TYPE ST_ITC_ZoneCommands :
(**************************************************************************************
 * 	Application		:	BoxControl Framework
 *	Revision		:	$Revision: 404529 $
 *	Revision date	:	$Date: 2018-04-23 08:21:38 +0200 (Mo., 23 Apr 2018) $
 *	Last changed by	:	$Author: b7bolm $
 *	URL				:	$URL: http://almscdc.swisslog.com/repo/SWPD/Development/BoxControlFramework/20_Release/trunk/01_Software/BCF/BCF/JumpStart/20_Product/10_App/12_E_Functions/10_Lib/10_Conv/01_DUTs/ST_ITC_ZoneCommands.TcDUT $
 *
 *	Purpose			:	Zone commands
 *
 * ------------------------------------------------------------------------------------
 *	Copyright Swisslog [IP AG], Switzerland. All rights reserved.
 * 
 * ------------------------------------------------------------------------------------
 *	
 * 	Revision History: 
 *
 * 	VERSION			DATE			INITIALS			DESCRIPTION
 *	0.1				01.01.2001		swl					Example
 *
 **************************************************************************************)	
STRUCT
	NoErrorReport				: BOOL; // Command to send a no error report 
	StatusReport				: BOOL; // Command to send a status report 
	ControlReport				: BOOL; // Command TO send a control report 
	TransportTaskCompleted		: BOOL; // Command to send a transport task report 
	PositionOccupied			: BOOL; // Command to send a position occupied report 
	PositionCleared				: BOOL; // Command to send a position cleared report 
	IdentificationReport		: BOOL; // Command to send an identification point report
END_STRUCT
END_TYPE

(* stored: Version 1.1.0.1, ProductVersion 3.1.4022.12
   DUT ST_ITC_ZoneCommands: Id {829b1abe-3b5d-491c-ad22-8873ebaa701e} *)
